// TIA Portal V20 export
TYPE "type_emRelations_em10_cmStatus"
// stored: Access Published, Namespace Unit1
   STRUCT
      LaserMarkJRDetect : "LBC_typeDigitalSignalControlNode";
      LaserMarkStageLiftUpDown : "LBC_typeTwoWayActuatorControlNode";
      LaserMarkCoverUpDown : "LBC_typeTwoWayActuatorControlNode";
      LaserMarkControl : "LER_typeLaserMarkControlNode";
      QrFixReaderControl : "LER_typeSRX300ControlNode";
   END_STRUCT;
END_TYPE
